FUNCTION_BLOCK Execute_State_Sample  IMPLEMENTS ITF_State
VAR_INPUT
END_VAR
VAR_OUTPUT
END_VAR
VAR
	pPML_Base : POINTER TO PML_StatePattern_Base;
	_stateMachine : IPmlStateMachine;
	bShutdown : BOOL;	
END_VAR

METHOD Cycle : BOOL
VAR_INPUT
END_VAR
IF bShutdown THEN
	pPML_Base^.SetState(pPML_Base^.aborting);
	_stateMachine.PmlStateCommand(Command := E_PMLCommand.ePMLCommand_Abort);
END_IF
END_METHOD

METHOD FB_init : BOOL
VAR_INPUT
	bInitRetains : BOOL; // if TRUE, the retain variables are initialized (warm start / cold start)
	bInCopyCode : BOOL;  // if TRUE, the instance afterwards gets moved into the copy code (online change)
	pPML_Base : POINTER TO PML_StatePattern_Base;
	statemachine : IPmlStateMachine;
END_VAR
_stateMachine := statemachine;
THIS^.pPML_Base := pPML_Base;
END_METHOD

END_FUNCTION_BLOCK

(* stored: Version 1.1.0.1, ProductVersion 3.1.4024.12
   POU Execute_State_Sample: Id {a87d20ee-0a99-4a25-9138-39db5a008f03}, SpecialFunc None
   Method Cycle: Id {b098cacd-f51d-4a54-a2b6-7608fd53a569}
   Method FB_init: Id {42ba6882-4e6a-428e-8cf7-579a088ff702} *)
